INTERFACE I_Cylinder EXTENDS I_CylinderCommand, I_CylinderStatus, I_Component, I_TaskResult, I_Resettable

{attribute 'monitoring' := 'call'}
PROPERTY ExtendTimeout : TIME
GET
END_GET
SET
END_SET
END_PROPERTY

{attribute 'monitoring' := 'call'}
PROPERTY RetractTimeout : TIME
GET
END_GET
SET
END_SET
END_PROPERTY

END_INTERFACE

(* stored: Version 1.1.0.1, ProductVersion 3.1.4026.18
   Itf I_Cylinder: Id {88e118d9-49e1-4dc0-8087-e4cfc085c749}
   Property ExtendTimeout: Id {941e9be6-201c-4da0-a311-088a51d256e9}
   Get Get: Id {28cc2abc-3e8b-4ec3-8a28-bb0523fcffa4}
   Set Set: Id {2c8551b4-5685-4459-8578-50a791e10694}
   Property RetractTimeout: Id {00d4233f-0041-4e77-be78-6dc82595dec7}
   Get Get: Id {8fd610f7-8b94-40ff-af29-6a103740d1a7}
   Set Set: Id {36d3d55f-890b-4ed4-90db-6863bbc16195} *)
